// Check if an external error is stored
ELSIF FunctionData.ErrorData.ExternalError.ErrorType > E_ErrorType.NO_ERROR_PENDING THEN
	// If error type has changed - its gone or type has changed
	IF FunctionData.ErrorData.ExternalError.ErrorType <> 
	   FunctionData.ErrorData.Error.ErrorType THEN
	   
		// If the stored error type was "ERROR"
		IF FunctionData.ErrorData.Error.ErrorType = E_ErrorType.ERROR
			OR FunctionData.ErrorData.Error.ErrorType = E_ErrorType.WARNING THEN
			// Send error is gone
			ITC.FunctionITC.Commands.NoErrorReport := TRUE;
		END_IF
		
		// Reset Message
		FunctionData.ErrorData.Error.ResetError 	:= FALSE;
		FunctionData.ErrorData.Error.ErrorType 	:= NO_ERROR_PENDING;
		FunctionData.ErrorData.Error.ErrorCode.Conv:= E_ErrorConv.NO_ERROR_CODE;
		FunctionData.ErrorData.Error.ErrorParam 	:= '';
	END_IF
END_IF

(**************************************************************************************************************
   Check for new or higher prioritized message
***************************************************************************************************************)
// Loop trough all error sets errors 
FOR mIdx := 1 TO NUMBER_OF_ERROR_SETS DO
	// Detect new or higher prioritized error message
	IF FunctionData.ErrorData.ErrorDataSet[mIdx].ErrorType > 
       FunctionData.ErrorData.Error.ErrorType THEN
		// Store index of current data set
		FunctionData.ErrorData.DataSetIdx := mIdx;
		
		// Update error
		FunctionData.ErrorData.Error.ErrorCode.Conv := FunctionData.ErrorData.ErrorDataSet[mIdx].ErrorCode.Conv;
		FunctionData.ErrorData.Error.ErrorParam := FunctionData.ErrorData.ErrorDataSet[mIdx].ErrorParam;
		FunctionData.ErrorData.Error.ErrorType := FunctionData.ErrorData.ErrorDataSet[mIdx].ErrorType;
		
		// Send Report
		ITC.FunctionITC.Commands.StatusReport := TRUE;
	END_IF
	
	// Check is an error is ongoing and a reset command is set
	IF FunctionData.ErrorData.Error.ResetError AND 
       FunctionData.ErrorData.ErrorDataSet[mIdx].ErrorType <> NO_ERROR_PENDING THEN
	   
		// Reset current error data set
		FunctionData.ErrorData.ErrorDataSet[mIdx].ResetError := TRUE;
	END_IF
END_FOR


// Check external error slot
IF FunctionData.ErrorData.ExternalError.ErrorType > FunctionData.ErrorData.Error.ErrorType THEN

	// Reset lower prioritized previous errors
	mDataSetIdx := 0;
	
	// Update error
	FunctionData.ErrorData.Error.ErrorCode.Conv := FunctionData.ErrorData.ExternalError.ErrorCode.Conv;
	FunctionData.ErrorData.Error.ErrorParam := FunctionData.ErrorData.ExternalError.ErrorParam;
	FunctionData.ErrorData.Error.ErrorType := FunctionData.ErrorData.ExternalError.ErrorType;

	// Send Report
	ITC.FunctionITC.Commands.StatusReport := TRUE;
END_IF

// Check is an external error is ongoing and a reset command is set
IF FunctionData.ErrorData.Error.ResetError AND 
   FunctionData.ErrorData.ExternalError.ErrorType <> NO_ERROR_PENDING THEN
   
	// Reset current error data set
	FunctionData.ErrorData.ExternalError.ResetError := TRUE;
END_IF


// If reset command is set
IF FunctionData.ErrorData.Error.ResetError THEN
	// If the stored error type was "ERROR"
	IF FunctionData.ErrorData.Error.ErrorType = E_ErrorType.ERROR THEN
		// Send error is gone
		ITC.FunctionITC.Commands.NoErrorReport := TRUE;
	END_IF
	
	// Reset stored data index
	FunctionData.ErrorData.DataSetIdx := 0;	

	// Reset Message
	FunctionData.ErrorData.Error.ResetError 	:= FALSE;
	FunctionData.ErrorData.Error.ErrorType 	:= NO_ERROR_PENDING;
	FunctionData.ErrorData.Error.ErrorCode.Conv:= E_ErrorConv.NO_ERROR_CODE;
	FunctionData.ErrorData.Error.ErrorParam 	:= '';
END_IF


(**************************************************************************************************************
   Function error state
***************************************************************************************************************)
// If function is in error state
IF FunctionData.ErrorData.Error.ErrorType = E_ErrorType.ERROR THEN
	// Set error state - ERROR
	FunctionData.ErrorData.ErrorState := E_ErrorState.ERROR;
	
// If function is in warning state
ELSIF FunctionData.ErrorData.Error.ErrorType = E_ErrorType.WARNING THEN
	// Set error state - WARNING
	FunctionData.ErrorData.ErrorState := E_ErrorState.WARNING;

// If function has no error or an info is pending
ELSIF FunctionData.ErrorData.Error.ErrorType = E_ErrorType.NO_ERROR_PENDING OR 
	  FunctionData.ErrorData.Error.ErrorType = E_ErrorType.INFO  THEN
	// Set error state - Operational
	FunctionData.ErrorData.ErrorState := E_ErrorState.OPERATIONAL;

ELSE
	// Otherwise -> Unknown
	FunctionData.ErrorData.ErrorState := E_ErrorState.UNKNOWN;
END_IF
END_METHOD

///Monitor zone errors - Verify error handling and report new errors.
METHOD PROTECTED M_MonitorZoneErrors : BOOL
(**************************************************************************************
 * Application   : BoxControl Framework
 * Revision date : $Date: 2021-04-09 16:13:33 +0200 (fre, 09 apr 2021) $
 * Author        : CDC
 * ------------------------------------------------------------------------------------
 * © Swisslog AG * Swisslog is not liable for any usage of this source code that is not agreed
 * on between Swisslog and the other party. The mandatory legal liability remains * unaffected.
 * ------------------------------------------------------------------------------------
 * Project revision history:
 *
 * VERSION DATE         INITIALS     DESCRIPTION
 * 0.0     DD.MM.YYYY   name       	 explain customized modifications
 *
 **************************************************************************************)
VAR
	mDataSetIdx				: INT; // Temporary data set index
	mIdx					: INT; // Iterator
	mZoneIdx				: INT; // Iterator through all zones
END_VAR
// Initialize
FunctionData.ErrorData.ZoneErrorPending := FALSE;

(**************************************************************************************************************
   Zone error handling
***************************************************************************************************************)
// Go through all zones
FOR mZoneIdx := 1 TO SettingsFunction.NumberOfZones DO
	
	// Store current zone data set index
	mDataSetIdx := ZoneData[mZoneIdx].ErrorData.DataSetIdx;
	
	// Check if an error is stored
	IF mDataSetIdx > 0 THEN
		
		// If error type has changed - its gone or type has changed
		IF ZoneData[mZoneIdx].ErrorData.ErrorDataSet[mDataSetIdx].ErrorType <> 
           ZoneData[mZoneIdx].ErrorData.Error.ErrorType THEN
			
			// If the stored error type was "ERROR"
			IF ZoneData[mZoneIdx].ErrorData.Error.ErrorType = E_ErrorType.ERROR
			   OR ZoneData[mZoneIdx].ErrorData.Error.ErrorType = E_ErrorType.WARNING  THEN
				// Send error is gone
				ITC.ZoneITC[mZoneIdx].Commands.NoErrorReport := TRUE;
			END_IF
			
			// Reset stored data index
			ZoneData[mZoneIdx].ErrorData.DataSetIdx := 0;		
					
			// Reset Message
			ZoneData[mZoneIdx].ErrorData.Error.ResetError := FALSE;
			ZoneData[mZoneIdx].ErrorData.Error.ErrorType := NO_ERROR_PENDING;
			ZoneData[mZoneIdx].ErrorData.Error.ErrorCode.Conv := E_ErrorConv.NO_ERROR_CODE;
			ZoneData[mZoneIdx].ErrorData.Error.ErrorParam := '';
		END_IF
		// Check if an external error is stored
	ELSIF ZoneData[mZoneIdx].ErrorData.ExternalError.ErrorType > E_ErrorType.NO_ERROR_PENDING THEN
		// If error type has changed - its gone or type has changed
		IF ZoneData[mZoneIdx].ErrorData.ExternalError.ErrorType <> 
		   ZoneData[mZoneIdx].ErrorData.Error.ErrorType THEN
		   
			// If the stored error type was "ERROR"
			IF ZoneData[mZoneIdx].ErrorData.Error.ErrorType = E_ErrorType.ERROR 
			   OR ZoneData[mZoneIdx].ErrorData.Error.ErrorType = E_ErrorType.WARNING THEN
				// Send error is gone
				ITC.ZoneITC[mZoneIdx].Commands.NoErrorReport := TRUE;
			END_IF
			
			// Reset Message
			ZoneData[mZoneIdx].ErrorData.Error.ResetError 		:= FALSE;
			ZoneData[mZoneIdx].ErrorData.Error.ErrorType 		:= NO_ERROR_PENDING;
			ZoneData[mZoneIdx].ErrorData.Error.ErrorCode.Conv	:= E_ErrorConv.NO_ERROR_CODE;
			ZoneData[mZoneIdx].ErrorData.Error.ErrorParam 		:= '';
		END_IF
	END_IF
	
	(**************************************************************************************************************
	   Check for new or higher prioritized message
	***************************************************************************************************************)
	
	// Loop trough all errors 
	FOR mIdx := 1 TO NUMBER_OF_ERROR_SETS DO
		// Detect new or higher prioritized error message
		IF ZoneData[mZoneIdx].ErrorData.ErrorDataSet[mIdx].ErrorType > 
		   ZoneData[mZoneIdx].ErrorData.Error.ErrorType THEN
			
			// Store index of current data set
			ZoneData[mZoneIdx].ErrorData.DataSetIdx := mIdx;
			
			// Update error
			ZoneData[mZoneIdx].ErrorData.Error.ErrorCode.Conv := ZoneData[mZoneIdx].ErrorData.ErrorDataSet[mIdx].ErrorCode.Conv;
			ZoneData[mZoneIdx].ErrorData.Error.ErrorParam := ZoneData[mZoneIdx].ErrorData.ErrorDataSet[mIdx].ErrorParam;
			ZoneData[mZoneIdx].ErrorData.Error.ErrorType := ZoneData[mZoneIdx].ErrorData.ErrorDataSet[mIdx].ErrorType;
			
			// Send Report
			ITC.ZoneITC[mZoneIdx].Commands.StatusReport := TRUE;
		END_IF
		
		// Check is an error is ongoing and a reset command is set
		IF ZoneData[mZoneIdx].ErrorData.Error.ResetError AND 
		   ZoneData[mZoneIdx].ErrorData.ErrorDataSet[mIdx].ErrorType <> NO_ERROR_PENDING THEN
		   
			// Reset current error data set
			ZoneData[mZoneIdx].ErrorData.ErrorDataSet[mIdx].ResetError := TRUE;
		END_IF
	END_FOR
	
	// Check external error slot
	IF ZoneData[mZoneIdx].ErrorData.ExternalError.ErrorType > ZoneData[mZoneIdx].ErrorData.Error.ErrorType THEN
		// Reset lower prioritized previous errors
		mDataSetIdx := 0;
		
		// Update error
		ZoneData[mZoneIdx].ErrorData.Error.ErrorCode.Conv := ZoneData[mZoneIdx].ErrorData.ExternalError.ErrorCode.Conv;
		ZoneData[mZoneIdx].ErrorData.Error.ErrorParam := ZoneData[mZoneIdx].ErrorData.ExternalError.ErrorParam;
		ZoneData[mZoneIdx].ErrorData.Error.ErrorType := ZoneData[mZoneIdx].ErrorData.ExternalError.ErrorType;
	
		// Send Report
		ITC.ZoneITC[mZoneIdx].Commands.StatusReport := TRUE;
	END_IF
	
	// Check is an external error is ongoing and a reset command is set
	IF ZoneData[mZoneIdx].ErrorData.Error.ResetError AND 
	   ZoneData[mZoneIdx].ErrorData.ExternalError.ErrorType <> NO_ERROR_PENDING THEN
	   
		// Reset current error data set
		ZoneData[mZoneIdx].ErrorData.ExternalError.ResetError := TRUE;
	END_IF
	
	// If reset command is set
	IF ZoneData[mZoneIdx].ErrorData.Error.ResetError THEN

		// If the stored error type was "ERROR"
		IF ZoneData[mZoneIdx].ErrorData.Error.ErrorType = E_ErrorType.ERROR THEN
			// Send error is gone
			ITC.ZoneITC[mZoneIdx].Commands.NoErrorReport := TRUE;
		END_IF
		
		// Reset stored data index
		ZoneData[mZoneIdx].ErrorData.DataSetIdx := 0;	
	
		// Reset Message
		ZoneData[mZoneIdx].ErrorData.Error.ResetError 	:= FALSE;
		ZoneData[mZoneIdx].ErrorData.Error.ErrorType := NO_ERROR_PENDING;
		ZoneData[mZoneIdx].ErrorData.Error.ErrorCode.Conv := E_ErrorConv.NO_ERROR_CODE;
		ZoneData[mZoneIdx].ErrorData.Error.ErrorParam 	:= '';
	END_IF
	
	
	(**************************************************************************************************************
	   zone error state
	***************************************************************************************************************)
	
	// If function is in error state
	IF ZoneData[mZoneIdx].ErrorData.Error.ErrorType = E_ErrorType.ERROR THEN
		// Set error state - ERROR
		ZoneData[mZoneIdx].ErrorData.ErrorState := E_ErrorState.ERROR;
		
	// If function is in warning state
	ELSIF ZoneData[mZoneIdx].ErrorData.Error.ErrorType = E_ErrorType.WARNING THEN
		// Set error state - WARNING
		ZoneData[mZoneIdx].ErrorData.ErrorState := E_ErrorState.WARNING;
	
	// If function has no error or an info is pending
	ELSIF ZoneData[mZoneIdx].ErrorData.Error.ErrorType = E_ErrorType.NO_ERROR_PENDING OR 
		  ZoneData[mZoneIdx].ErrorData.Error.ErrorType = E_ErrorType.INFO  THEN
		// Set error state - Operational
		ZoneData[mZoneIdx].ErrorData.ErrorState := E_ErrorState.OPERATIONAL;
	
	ELSE
		// Otherwise -> Unknown
		ZoneData[mZoneIdx].ErrorData.ErrorState := E_ErrorState.UNKNOWN;
	END_IF
	
	(**************************************************************************************************************
	   Inform function about zone error state
	***************************************************************************************************************)
	FunctionData.ErrorData.ZoneErrorPending := FunctionData.ErrorData.ZoneErrorPending OR
															ZoneData[mZoneIdx].ErrorData.Error.ErrorType = E_ErrorType.ERROR;
END_FOR
END_METHOD

METHOD M_MoveTU_DataIndex : DINT;
(**************************************************************************************
 * 	Application		:	BoxControl Framework
 *	Revision		:	$Revision: 475069 $
 *	Revision date	:	$Date: 2021-04-09 16:13:33 +0200 (fre, 09 apr 2021) $
 *	Last changed by	:	$Author: d7mangc $
 *	URL				:	$URL: http://almscdc.swisslog.com/repo/SWPD/Development/BoxControlFramework/20_Release/tags/R1.12.0/01_Software/BCF/BCF/JumpStart/20_Product/10_BCF/11_Conv/12_E_Functions/FB_FunctionConv.TcPOU $
 *
 *	Purpose			:	Moves the TU-data index from zone to zone and updates the states.
 *
 * ------------------------------------------------------------------------------------
 *	Copyright Swisslog [IP AG], Switzerland. All rights reserved.
 * 
 * ------------------------------------------------------------------------------------
 *	
 * 	Revision History: 
 *
 * 	VERSION			DATE			INITIALS			DESCRIPTION
 *	0.1				01.01.2001		swl					Example
 *
 **************************************************************************************)
VAR_INPUT
	mZoneNumber : INT;
END_VAR
// Return current TU data index
M_MoveTU_dataIndex := ZoneData[mZoneNumber].TransportControlData.TU_DataIndex;
// Update last TU data index
ZoneData[mZoneNumber].TransportControlData.LastTU_DataIndex := M_MoveTU_dataIndex;
// Delete current TU data index
ZoneData[mZoneNumber].TransportControlData.TU_DataIndex := 0;
// Reset data present flag
ZoneData[mZoneNumber].TransportControlData.DataPresent := FALSE;
// Update number of present TUs 
IF ZoneData[mZoneNumber].TransportControlData.NumberOfPresentTUs > 0 THEN
	ZoneData[mZoneNumber].TransportControlData.NumberOfPresentTUs := ZoneData[mZoneNumber].TransportControlData.NumberOfPresentTUs -1;
END_IF


// BCFD-11639 - POR0 - Position Cleared Report sent without TU-ID	
// included in BCF 1.16
// Save data from the last TU for the position clear report
M_SaveDataTU_ZoneLeft (mZoneNumber, M_MoveTU_dataIndex);
END_METHOD

METHOD PROTECTED M_MsgHandlerZone : BOOL
(**************************************************************************************
 * 	Application		:	BoxControl Framework
 *	Revision		:	$Revision: 475069 $
 *	Revision date	:	$Date: 2021-04-09 16:13:33 +0200 (fre, 09 apr 2021) $
 *	Last changed by	:	$Author: d7mangc $
 *	URL				:	$URL: http://almscdc.swisslog.com/repo/SWPD/Development/BoxControlFramework/20_Release/tags/R1.12.0/01_Software/BCF/BCF/JumpStart/20_Product/10_BCF/11_Conv/12_E_Functions/FB_FunctionConv.TcPOU $
 *
 *	Purpose			:	Function zone ITC out interface
 *						Handles internally set ITC commands.
 *
 * ------------------------------------------------------------------------------------
 *	Copyright Swisslog [IP AG], Switzerland. All rights reserved.
 * 
 * ------------------------------------------------------------------------------------
 *	
 * 	Revision History: 
 *
 * 	VERSION			DATE			INITIALS			DESCRIPTION
 *	0.1				01.01.2001		swl					Example
 *
 **************************************************************************************)
VAR_INPUT
	mZoneNumber			: INT; // Zone number	
END_VAR

VAR
	mTU_DataIndex		: DINT;
	mIdx				: INT; // Iterator
END_VAR

// If a valid zone is configured
IF mZoneNumber > 0 AND mZoneNumber <= SettingsFunction.NumberOfZones THEN
	
	// TU data index
	mTU_DataIndex := ZoneData[mZoneNumber].TransportControlData.TU_DataIndex;

	(*******************************************************************************
		Transport Task Complete - TTC
	********************************************************************************)
	// If data are present on zone
	IF ZoneData[mZoneNumber].TransportControlData.DataPresent THEN
		
		// Go through all destination of the TU
		FOR mIdx := 1 TO TU_DataTable[mTU_DataIndex].DataSet.NumberOfDest DO
			// Check destination
			IF TU_DataTable[mTU_DataIndex].Destination[mIdx].eFunctionNumber = SettingsFunction.eFunctionNumber AND
			   TU_DataTable[mTU_DataIndex].Destination[mIdx].ZoneNumber =	mZoneNumber THEN
			   
			   	// When a TTC is requested when data are present
				IF SettingsFunction.Zone[mZoneNumber].SendTransportTaskCompleted AND 
				   NOT ITC.ZoneITC[mZoneNumber].Flags.TransportTaksCompleteSent THEN
					// Send telegram & flag
					ITC.ZoneITC[mZoneNumber].Commands.TransportTaskCompleted := TRUE;
					ITC.ZoneITC[mZoneNumber].Flags.TransportTaksCompleteSent := TRUE;
				END_IF
				
				// When a TTC is requested when data are present and location occupied
				IF SettingsFunction.Zone[mZoneNumber].SendTransportTaskCompletedOcc AND 
				   ZoneData[mZoneNumber].TransportControlData.Occupied AND
				   NOT ITC.ZoneITC[mZoneNumber].Flags.TransportTaksCompleteOccSent THEN
					// Send telegram & flag
					ITC.ZoneITC[mZoneNumber].Commands.TransportTaskCompleted := TRUE;
					ITC.ZoneITC[mZoneNumber].Flags.TransportTaksCompleteOccSent := TRUE;
				END_IF
				
				// When no TTC is configured or already sent - Reset destination
				IF (NOT SettingsFunction.Zone[mZoneNumber].SendTransportTaskCompleted OR ITC.ZoneITC[mZoneNumber].Flags.TransportTaksCompleteSent) AND
				   (NOT SettingsFunction.Zone[mZoneNumber].SendTransportTaskCompletedOcc OR ITC.ZoneITC[mZoneNumber].Flags.TransportTaksCompleteOccSent) THEN
					// Delete destination
					F_DeleteDestination(eFunctionNumber := SettingsFunction.eFunctionNumber, ZoneNumber := mZoneNumber);
				   EXIT;
				END_IF
			END_IF
		END_FOR
	ELSE
		// Reset flags
		ITC.ZoneITC[mZoneNumber].Flags.TransportTaksCompleteSent := FALSE;
		ITC.ZoneITC[mZoneNumber].Flags.TransportTaksCompleteOccSent := FALSE;
	END_IF
	
	(*******************************************************************************
		Position Clear Report 
	********************************************************************************)
	// When a position clear report is requested 
	IF SettingsFunction.Zone[mZoneNumber].SendPositionClear THEN 
		// Is corresponding function started
	   	IF FunctionData.OperationState.eState = E_PositionState.STARTED THEN
			// Is zone free
			IF NOT ZoneData[mZoneNumber].TransportControlData.Occupied THEN
				// And not sent so far
				IF NOT ITC.ZoneITC[mZoneNumber].Flags.PositionClearSent THEN
					// Send telegram & flag
					ITC.ZoneITC[mZoneNumber].Commands.PositionCleared := TRUE;
					ITC.ZoneITC[mZoneNumber].Flags.PositionClearSent := TRUE;
				END_IF
			ELSE
				// Reset flag
				ITC.ZoneITC[mZoneNumber].Flags.PositionClearSent := FALSE;
			END_IF
		END_IF
	ELSE
		// Reset flag
		ITC.ZoneITC[mZoneNumber].Flags.PositionClearSent := FALSE;
	END_IF
	
	(*******************************************************************************
		Position Occupied Report 
	********************************************************************************)
	// When a position occupied report is requested 
	IF SettingsFunction.Zone[mZoneNumber].SendPositionOccupied THEN 
		// Is corresponding function started
	   	IF FunctionData.OperationState.eState = E_PositionState.STARTED THEN
			// Is zone occupied
			IF ZoneData[mZoneNumber].TransportControlData.Occupied THEN
				// And not sent so far
				IF NOT ITC.ZoneITC[mZoneNumber].Flags.PositionOccupiedSent THEN
					// Send telegram & flag
					ITC.ZoneITC[mZoneNumber].Commands.PositionOccupied := TRUE;
					ITC.ZoneITC[mZoneNumber].Flags.PositionOccupiedSent := TRUE;
				END_IF
			ELSE
				// Reset flag
				ITC.ZoneITC[mZoneNumber].Flags.PositionOccupiedSent := FALSE;
			END_IF
		END_IF
	ELSE
		// Reset flag
		ITC.ZoneITC[mZoneNumber].Flags.PositionOccupiedSent := FALSE;
	END_IF
	
	(*******************************************************************************
		Identification Point Report 
	********************************************************************************)
	// When a identification report is requested 
	IF SettingsFunction.Zone[mZoneNumber].SendIdentificationReport THEN 
		// When data are present
		IF ZoneData[mZoneNumber].TransportControlData.DataPresent THEN
			// If the zone is occupied and no add-on is assigned or data ready from all addons is set
			// the telegramm can be triggered.
			IF ZoneData[mZoneNumber].TransportControlData.Occupied THEN 
				IF ZoneData[mZoneNumber].AddOn.NoAddons OR ZoneData[mZoneNumber].AddOn.Orders.DataReady THEN
					// And not sent so far
					IF NOT ITC.ZoneITC[mZoneNumber].Flags.IdentificationReportSent THEN
						// Send telegram & flag
						ITC.ZoneITC[mZoneNumber].Commands.IdentificationReport := TRUE;
						ITC.ZoneITC[mZoneNumber].Flags.IdentificationReportSent := TRUE;
					END_IF
				END_IF
			ELSE
				// Reset flag
				ITC.ZoneITC[mZoneNumber].Flags.IdentificationReportSent := FALSE;
			END_IF
		ELSE
			// Reset flag
			ITC.ZoneITC[mZoneNumber].Flags.IdentificationReportSent := FALSE;
		END_IF
	ELSE
		// Reset flag
		ITC.ZoneITC[mZoneNumber].Flags.IdentificationReportSent := FALSE;
	END_IF
END_IF
END_METHOD

METHOD M_PreInit : BOOL
(**************************************************************************************
 * 	Application		:	BoxControl Framework
 *	Revision		:	$Revision: 475069 $
 *	Revision date	:	$Date: 2021-04-09 16:13:33 +0200 (fre, 09 apr 2021) $
 *	Last changed by	:	$Author: d7mangc $
 *	URL				:	$URL: http://almscdc.swisslog.com/repo/SWPD/Development/BoxControlFramework/20_Release/tags/R1.12.0/01_Software/BCF/BCF/JumpStart/20_Product/10_BCF/11_Conv/12_E_Functions/FB_FunctionConv.TcPOU $
 *
 *	Purpose			:	Preinitialize 
 *						Clears values and load settings
 *
 * ------------------------------------------------------------------------------------
 *	Copyright Swisslog [IP AG], Switzerland. All rights reserved.
 * 
 * ------------------------------------------------------------------------------------
 *	
 * 	Revision History: 
 *
 * 	VERSION			DATE			INITIALS			DESCRIPTION
 *	0.1				01.01.2001		swl					Example
 *
 **************************************************************************************)
VAR
	eFunctionNumber	: E_FunctionNumber; 
	eElementNumber	: E_ElementNumber;
END_VAR
(**************************************************************************************
   		Unregister
***************************************************************************************)	
// If Addon function link has changed
IF SettingsFunction.FunctionLink.eFunctionNumber <> ConfigFunction.FunctionLink.eFunctionNumber AND
   SettingsFunction.FunctionLink.eFunctionNumber > E_FunctionNumber.F_BEGIN_FUNCTION THEN
   
	// Close old addon link
	eFunctionNumber := SettingsFunction.FunctionLink.eFunctionNumber;
	
	// Is this reference valid
	IF __ISVALIDREF(FunctionRegistry[eFunctionNumber].rFunction) THEN
		// Close AddOn link
		FunctionRegistry[eFunctionNumber].rFunction.M_CloseAddOnLink(eAddOnNumber := SettingsFunction.eFunctionNumber);
	END_IF
END_IF

// If element link has changed
IF SettingsFunction.eElementLink <> ConfigFunction.eElementLink AND 
   SettingsFunction.eElementLink > E_ElementNumber.E_BEGIN_ELEMENT THEN
	// Close old element link
	eElementNumber := SettingsFunction.eElementLink;
	
	// Is reference valid
	IF __ISVALIDREF(ElementRegistry[eElementNumber].rElement) THEN
		// Unregister function in element
		ElementRegistry[eElementNumber].rElement.M_CloseElementLink(SettingsFunction.eFunctionNumber);
	END_IF
END_IF


// Clear previous and next function
FunctionInterface.In.ePrevFunctionNumber := E_FunctionNumber.F_BEGIN_FUNCTION;
FunctionInterface.In.eNextFunctionNumber := E_FunctionNumber.F_BEGIN_FUNCTION;


(**************************************************************************************
	Load 
***************************************************************************************)
SettingsFunction := ConfigFunction;
END_METHOD

METHOD PROTECTED M_ProcessAddOns
(**************************************************************************************
 * 	Application		:	BoxControl Framework
 *	Revision		:	$Revision: 475069 $
 *	Revision date	:	$Date: 2021-04-09 16:13:33 +0200 (fre, 09 apr 2021) $
 *	Last changed by	:	$Author: d7mangc $
 *	URL				:	$URL: http://almscdc.swisslog.com/repo/SWPD/Development/BoxControlFramework/20_Release/tags/R1.12.0/01_Software/BCF/BCF/JumpStart/20_Product/10_BCF/11_Conv/12_E_Functions/FB_FunctionConv.TcPOU $
 *
 *	Purpose			:	Process AddOns
 *
 * ------------------------------------------------------------------------------------
 *	Copyright Swisslog [IP AG], Switzerland. All rights reserved.
 * 
 * ------------------------------------------------------------------------------------
 *	
 * 	Revision History: 
 *
 * 	VERSION			DATE			INITIALS			DESCRIPTION
 *	0.1				01.01.2001		swl					Example
 *
 **************************************************************************************)
VAR
  mIdx             : INT; // Iterator
  mZoneNumber      : INT; // Zone number
  mTU_DataIndexNew : DINT; // TU data index new
  mTU_DataIndexOld : DINT; // TU data index old
  mSummary         : ST_AddOnOrders;
END_VAR
// Initialize var
mSummary.Enable         	:= TRUE;
mSummary.EnableHandover 	:= TRUE;
mSummary.EnableTakeover 	:= TRUE;
mSummary.DataReady      	:= TRUE;
mSummary.TU_DataIndex   	:= 0;
mSummary.EnableSimultaneousTransport := FALSE;
mSummary.UseOwnSensor 		:= FALSE;
mSummary.AddOnSensor 		:= FALSE;
mSummary.AllowDriveTakeover := FALSE;
mSummary.AllowDriveHandover := FALSE;

// Initialize all zones
FOR mIdx := 1 TO SettingsFunction.NumberOfZones DO
	ZoneData[mIdx].AddOn.NoAddons := TRUE;
	ZoneData[mIdx].AddOn.Orders := mSummary;
END_FOR

// Initialize function
FunctionData.AddOn.NoAddons := TRUE;
FunctionData.AddOn.Orders := mSummary;

// Build summary of all addon functions
FOR mIdx := 1 TO NUMBER_OF_ADDON_FUNCTIONS DO
	// If no addon is configured
	IF FunctionInterface.In.AddOnOrder[mIdx].eFunctionNumber = E_FunctionNumber.F_BEGIN_FUNCTION THEN
		// Exit loop
		EXIT;
	END_IF

	// Update summary from addon interface		   
	IF NOT FunctionInterface.In.AddOnOrder[mIdx].Orders.Enable THEN
		mSummary.Enable := FALSE;
	END_IF
	
	IF NOT FunctionInterface.In.AddOnOrder[mIdx].Orders.EnableHandover THEN
		mSummary.EnableHandover := FALSE;
	END_IF

	IF NOT FunctionInterface.In.AddOnOrder[mIdx].Orders.EnableTakeover  THEN
		mSummary.EnableTakeover := FALSE;
	END_IF

	IF NOT FunctionInterface.In.AddOnOrder[mIdx].Orders.DataReady THEN
		mSummary.DataReady := FALSE;
	END_IF
	
	IF NOT FunctionInterface.In.AddOnOrder[mIdx].Orders.DataValid THEN
		mSummary.DataValid := FALSE;
	END_IF
			
    IF FunctionInterface.In.AddOnOrder[mIdx].Orders.EnableSimultaneousTransport THEN
        mSummary.EnableSimultaneousTransport := TRUE;
	END_IF
    
    IF FunctionInterface.In.AddOnOrder[mIdx].Orders.AddOnSensor THEN
        mSummary.AddOnSensor := TRUE;
	END_IF
    
    IF FunctionInterface.In.AddOnOrder[mIdx].Orders.UseOwnSensor THEN
        mSummary.UseOwnSensor := TRUE;
	END_IF
    
    IF FunctionInterface.In.AddOnOrder[mIdx].Orders.AllowDriveTakeover THEN
        mSummary.AllowDriveTakeover := TRUE;
	END_IF
    
    IF FunctionInterface.In.AddOnOrder[mIdx].Orders.AllowDriveHandover THEN
        mSummary.AllowDriveHandover := TRUE;
	END_IF
    
	// Update zone or function data
	mZoneNumber := FunctionInterface.In.AddOnOrder[mIdx].ZoneNumber;
	
	IF mZoneNumber <= 0 THEN
		FunctionData.AddOn.NoAddons := FALSE;
		FunctionData.AddOn.Orders := mSummary;
	ELSIF mZoneNumber > SettingsFunction.NumberOfZones  THEN
		FunctionData.AddOn.NoAddons := FALSE;
		FunctionData.AddOn.Orders := mSummary;
	ELSE
		ZoneData[mZoneNumber].AddOn.NoAddons := FALSE;
		ZoneData[mZoneNumber].AddOn.Orders := mSummary;
	END_IF

	// If it is not a function type "Scanner"
	IF FunctionInterface.In.AddOnOrder[mIdx].eFunctionType <> E_FunctionType.Scanner THEN
		// Process next addon function
		CONTINUE;
	END_IF
	
	// Data ready is not set
	IF NOT FunctionInterface.In.AddOnOrder[mIdx].Orders.DataReady THEN
		// Process next addon function
		CONTINUE;
	END_IF
	
	// Data valid is not set
	IF NOT FunctionInterface.In.AddOnOrder[mIdx].Orders.DataValid THEN
		// Process next addon function
		CONTINUE;
	END_IF

	// Take over TU index
	mTU_DataIndexOld := ZoneData[mZoneNumber].TransportControlData.TU_DataIndex;
	mTU_DataIndexNew := FunctionInterface.In.AddOnOrder[mIdx].Orders.TU_DataIndex;
	ZoneData[mZoneNumber].AddOn.Orders.TU_DataIndex := mTU_DataIndexNew;

	// Update index only if takeover is active, feedin or multi TU	
	IF (ZoneData[mZoneNumber].TransportControlData.eTakeOverState = E_TakeOverState.ACTIVE AND
		(ZoneData[mZoneNumber].TransportControlData.eTransportState = E_TransportState.TAKEOVER OR
		 ZoneData[mZoneNumber].TransportControlData.eTransportState = E_TransportState.SIMULTANEOUS)) OR
	   ZoneData[mZoneNumber].TransportControlData.eTransportState = E_TransportState.FEEDIN OR
	   ZoneData[mZoneNumber].TransportControlData.eTransportState = E_TransportState.MULTI_TU THEN

		// When the conveyor do not have an index yet, just apply the scanner index
		IF mTU_DataIndexOld = 0 THEN
			// Create debug message	
			// '11-001-0095-01-1,  TU_DataIndex inserted by scanner,  TU_DataIndex = 5,  TuID = 000012345,  AssignmentID = 999999999 '
			DebugMsg := '';
			DebugMsg := CONCAT(DebugMsg, F_AddDividerToSisString(SettingsFunction.Zone[mZoneNumber].ZoneName));
			DebugMsg := CONCAT(DebugMsg, ',  TU_DataIndex inserted by scanner');
			DebugMsg := CONCAT(DebugMsg, F_CreateTU_DataString(TU_DataIndex:= mTU_DataIndexNew));
			fbDebugMsg.M_SendInfoMsg(DebugMsg);

			// Update TU data index
			ZoneData[mZoneNumber].TransportControlData.LastTU_DataIndex := mTU_DataIndexOld;
			ZoneData[mZoneNumber].TransportControlData.TU_DataIndex := mTU_DataIndexNew;
			ZoneData[mZoneNumber].TransportControlData.DataPresent := mTU_DataIndexNew <> 0;
	
			// Update current TU position
			TU_DataTable[mTU_DataIndexNew].CurrentFunctionNumber := SettingsFunction.eFunctionNumber;
			TU_DataTable[mTU_DataIndexNew].CurrentZoneNumber := mZoneNumber;

		// When a scanner provides an index unequal to the already existing conveyor index, takeover the scanner index.
		ELSIF mTU_DataIndexOld <> mTU_DataIndexNew THEN
			// Create debug message	
			// '11-001-0095-01-1,  TU_DataIndex overwritten by scanner (old/new),  TU_DataIndex = 5,  TuID = 000012345,  AssignmentID = 999999999,  TU_DataIndex = 9,  TuID = 000098765,  AssignmentID = 999999999',  Origin = 11-002-0125-02-2
			DebugMsg := '';
			DebugMsg := CONCAT(DebugMsg, F_AddDividerToSisString(SettingsFunction.Zone[mZoneNumber].ZoneName));
			DebugMsg := CONCAT(DebugMsg, ',  TU_DataIndex overwritten by scanner (old/new)');
			DebugMsg := CONCAT(DebugMsg, F_CreateTU_DataString(TU_DataIndex:= mTU_DataIndexOld));
			DebugMsg := CONCAT(DebugMsg, F_CreateTU_DataString(TU_DataIndex:= mTU_DataIndexNew));
			DebugMsg := CONCAT(DebugMsg, DebugTextBlocks.ORIGIN);
			DebugMsg := CONCAT(DebugMsg, F_GetFunctionName(
												eFunctionNumber := TU_DataTable[mTU_DataIndexNew].CurrentFunctionNumber,
												ZoneNumber := TU_DataTable[mTU_DataIndexNew].CurrentZoneNumber));
			fbDebugMsg.M_SendErrorMsg(DebugMsg);
												
			// If old TU data index is unknown, delete it from the table 
			IF TU_DataTable[mTU_DataIndexOld].TU_ID.ASCII = Conveyor.TU_ID_UNKNOWN THEN
				// debug message: '11-001-0095-01-1,  unknown old TU_DataIndex deleted,  TU_DataIndex = 5,  TuID = 000012345,  AssignmentID = 999999999'
				DebugMsg := '';
				DebugMsg := CONCAT(DebugMsg, F_AddDividerToSisString(SettingsFunction.Zone[mZoneNumber].ZoneName));
				DebugMsg := CONCAT(DebugMsg, ',  unknown old TU_DataIndex deleted');
				DebugMsg := CONCAT(DebugMsg, F_CreateTU_DataString(TU_DataIndex:= mTU_DataIndexOld));
				fbDebugMsg.M_SendErrorMsg(DebugMsg);
				// Delete data set
				F_DeleteTU_Data(TU_DataIndex := mTU_DataIndexOld,
                       			NoTTC := FALSE);
			END_IF

			// Update TU data index
			ZoneData[mZoneNumber].TransportControlData.LastTU_DataIndex := mTU_DataIndexOld;
			ZoneData[mZoneNumber].TransportControlData.TU_DataIndex := mTU_DataIndexNew;
			ZoneData[mZoneNumber].TransportControlData.DataPresent := mTU_DataIndexNew <> 0;
	
			// Update current TU position
			TU_DataTable[mTU_DataIndexNew].CurrentFunctionNumber := SettingsFunction.eFunctionNumber;
			TU_DataTable[mTU_DataIndexNew].CurrentZoneNumber := mZoneNumber;
		END_IF
					   
    	// Send ACK
		F_AckAddon(eFunctionNumber := FunctionInterface.In.AddOnOrder[mIdx].eFunctionNumber);
						
	ELSIF ZoneData[mZoneNumber].TransportControlData.eTransportState = E_TransportState.HANDOVER OR
		  ZoneData[mZoneNumber].TransportControlData.eTransportState = E_TransportState.OCCUPIED THEN
		 // Send ACK
		F_AckAddon(eFunctionNumber := FunctionInterface.In.AddOnOrder[mIdx].eFunctionNumber);
	END_IF
END_FOR
END_METHOD

METHOD M_ResetError : BOOL
(**************************************************************************************
 * 	Application		:	BoxControl Framework
 *	Revision		:	$Revision: 475069 $
 *	Revision date	:	$Date: 2021-04-09 16:13:33 +0200 (fre, 09 apr 2021) $
 *	Last changed by	:	$Author: d7mangc $
 *	URL				:	$URL: http://almscdc.swisslog.com/repo/SWPD/Development/BoxControlFramework/20_Release/tags/R1.12.0/01_Software/BCF/BCF/JumpStart/20_Product/10_BCF/11_Conv/12_E_Functions/FB_FunctionConv.TcPOU $
 *
 *	Purpose			:	Reset function or zone errors.
 *
 * ------------------------------------------------------------------------------------
 *	Copyright Swisslog [IP AG], Switzerland. All rights reserved.
 * 
 * ------------------------------------------------------------------------------------
 *	
 * 	Revision History: 
 *
 * 	VERSION			DATE			INITIALS			DESCRIPTION
 *	0.1				01.01.2001		swl					Example
 *
 **************************************************************************************)
VAR_INPUT
	mZoneNumber		: INT; // Zone number
	mResetAll		: BOOL; // Reset all
END_VAR

VAR
	mIdx			: INT; // Iterator
END_VAR
// Command is to reset all
IF mResetAll THEN
	// Go through all zones
	FOR mIdx := 1 TO NUMBER_OF_ZONES_PER_FUNCTION DO
		// If the zone is in error
		IF ZoneData[mIdx].ErrorData.Error.ErrorType  <> E_ErrorType.NO_ERROR_PENDING  THEN
			// Send reset
			ZoneData[mIdx].ErrorData.Error.ResetError := TRUE;
		END_IF
	END_FOR

	// If the function is in error
	IF FunctionData.ErrorData.Error.ErrorType  <> E_ErrorType.NO_ERROR_PENDING  THEN
		// Send reset
		FunctionData.ErrorData.Error.ResetError := TRUE;
	END_IF
	
// Command to reset a zone
ELSIF mZoneNumber > 0 AND mZoneNumber <= NUMBER_OF_ZONES_PER_FUNCTION THEN
	// If the zone is in error
	IF ZoneData[mZoneNumber].ErrorData.Error.ErrorType  <> E_ErrorType.NO_ERROR_PENDING  THEN
		// Send reset
		ZoneData[mZoneNumber].ErrorData.Error.ResetError := TRUE;
	END_IF
ELSE
	// If the function is in error
	IF FunctionData.ErrorData.Error.ErrorType  <> E_ErrorType.NO_ERROR_PENDING  THEN
		// Send reset
		FunctionData.ErrorData.Error.ResetError := TRUE;
	END_IF
END_IF

M_ResetError := TRUE;
END_METHOD

METHOD M_ResetExternalError : BOOL
(**************************************************************************************
 * 	Application		:	BoxControl Framework
 *	Revision		:	$Revision: 475069 $
 *	Revision date	:	$Date: 2021-04-09 16:13:33 +0200 (fre, 09 apr 2021) $
 *	Last changed by	:	$Author: d7mangc $
 *	URL				:	$URL: http://almscdc.swisslog.com/repo/SWPD/Development/BoxControlFramework/20_Release/tags/R1.12.0/01_Software/BCF/BCF/JumpStart/20_Product/10_BCF/11_Conv/12_E_Functions/FB_FunctionConv.TcPOU $
 *
 *	Purpose			:	Reset external error
 *						
 *
 * ------------------------------------------------------------------------------------
 *	Copyright Swisslog [IP AG], Switzerland. All rights reserved.
 * 
 * ------------------------------------------------------------------------------------
 *	
 * 	Revision History: 
 *
 * 	VERSION			DATE			INITIALS			DESCRIPTION
 *	0.1				01.01.2001		swl					Example
 *
 **************************************************************************************)
 VAR_INPUT
	mZoneNumber	: INT; // Related zone, 0 = Function itself
	mReset		: BOOL; // Force reset
END_VAR
// Initialize
M_ResetExternalError := FALSE;

IF mZoneNumber > 0 THEN
	// Reset error if ResetError command or reset command is set 
	IF ZoneData[mZoneNumber].ErrorData.ExternalError.ResetError OR mReset THEN
		// Clear error
		ZoneData[mZoneNumber].ErrorData.ExternalError.ResetError 		:= FALSE; 
		ZoneData[mZoneNumber].ErrorData.ExternalError.ErrorType 		:= NO_ERROR_PENDING;
		ZoneData[mZoneNumber].ErrorData.ExternalError.ErrorCode.Conv	:= E_ErrorConv.NO_ERROR_CODE;
		ZoneData[mZoneNumber].ErrorData.ExternalError.ErrorParam 		:= '';
		M_ResetExternalError 								:= TRUE;
	END_IF
ELSE
	// Reset error if ResetError command or reset command is set 
	IF FunctionData.ErrorData.ExternalError.ResetError OR mReset THEN
		// Clear error
		FunctionData.ErrorData.ExternalError.ResetError 	:= FALSE; 
		FunctionData.ErrorData.ExternalError.ErrorType 		:= NO_ERROR_PENDING;
		FunctionData.ErrorData.ExternalError.ErrorCode.Conv	:= E_ErrorConv.NO_ERROR_CODE;
		FunctionData.ErrorData.ExternalError.ErrorParam 	:= '';
		M_ResetExternalError 								:= TRUE;
	END_IF
END_IF
END_METHOD

METHOD PUBLIC M_SaveDataTU_ZoneLeft : BOOL
VAR_INPUT
	mZoneNumber		: INT;
    mTU_DataIndex	: DINT;
END_VAR

// BCFD-11639 - POR0 - Position Cleared Report sent without TU-ID	
// included in BCF 1.16

// Save data from the last TU for the position clear report
ZoneData[mZoneNumber].LastTUdata.AssignmentID	:= TU_DataTable[mTU_DataIndex].AssignmentID;
ZoneData[mZoneNumber].LastTUdata.TU_ID			:= TU_DataTable[mTU_DataIndex].TU_ID.ASCII;
ZoneData[mZoneNumber].LastTUdata.TU_Type		:= TU_DataTable[mTU_DataIndex].DataSet.TU_Type;
END_METHOD

METHOD M_SetEnableHandOver : BOOL
(**************************************************************************************
 * 	Application		:	BoxControl Framework
 *	Revision		:	$Revision: 475069 $
 *	Revision date	:	$Date: 2021-04-09 16:13:33 +0200 (fre, 09 apr 2021) $
 *	Last changed by	:	$Author: d7mangc $
 *	URL				:	$URL: http://almscdc.swisslog.com/repo/SWPD/Development/BoxControlFramework/20_Release/tags/R1.12.0/01_Software/BCF/BCF/JumpStart/20_Product/10_BCF/11_Conv/12_E_Functions/FB_FunctionConv.TcPOU $
 *
 *	Purpose			:	Initialize base functionality of function.
 *
 * ------------------------------------------------------------------------------------
 *	Copyright Swisslog [IP AG], Switzerland. All rights reserved.
 * 
 * ------------------------------------------------------------------------------------
 *	
 * 	Revision History: 
 *
 * 	VERSION			DATE			INITIALS			DESCRIPTION
 *	0.1				01.01.2001		swl					Example
 *
 **************************************************************************************)
VAR_INPUT
	mZoneNumber 	: INT; // Zone number
	mValue			: BOOL; // Set/reset value
END_VAR
// If zone number is valid
IF mZoneNumber > 0 AND mZoneNumber <= SettingsFunction.NumberOfZones THEN
	// Modify variable
	ZoneInterface[mZoneNumber].In.Enable.HandOver := mValue;
	M_SetEnableHandOver := TRUE;

// Otherwise requested index was not found
ELSE	
	DebugMsg := CONCAT('Requested zone not available: ', INT_TO_STRING(mZoneNumber));
	fbDebugMsg.M_SendErrorMsg(DebugMsg);
END_IF
END_METHOD

METHOD M_SetEnableTakeOver : BOOL
(**************************************************************************************
 * 	Application		:	BoxControl Framework
 *	Revision		:	$Revision: 475069 $
 *	Revision date	:	$Date: 2021-04-09 16:13:33 +0200 (fre, 09 apr 2021) $
 *	Last changed by	:	$Author: d7mangc $
 *	URL				:	$URL: http://almscdc.swisslog.com/repo/SWPD/Development/BoxControlFramework/20_Release/tags/R1.12.0/01_Software/BCF/BCF/JumpStart/20_Product/10_BCF/11_Conv/12_E_Functions/FB_FunctionConv.TcPOU $
 *
 *	Purpose			:	Initialize base functionality of function.
 *
 * ------------------------------------------------------------------------------------
 *	Copyright Swisslog [IP AG], Switzerland. All rights reserved.
 * 
 * ------------------------------------------------------------------------------------
 *	
 * 	Revision History: 
 *
 * 	VERSION			DATE			INITIALS			DESCRIPTION
 *	0.1				01.01.2001		swl					Example
 *
 **************************************************************************************)
VAR_INPUT
	mZoneNumber 	: INT; // Zone number
	mValue			: BOOL; // Set/reset value
END_VAR
// If zone number is valid
IF mZoneNumber > 0 AND mZoneNumber <= SettingsFunction.NumberOfZones THEN
	// Modify variable
	ZoneInterface[mZoneNumber].In.Enable.TakeOver := mValue;
	M_SetEnableTakeOver := TRUE;

// Otherwise requested index was not found
ELSE	
	DebugMsg := CONCAT('Requested zone not available: ', INT_TO_STRING(mZoneNumber));
	fbDebugMsg.M_SendErrorMsg(DebugMsg);
END_IF
END_METHOD

METHOD M_SetEnableTransport : BOOL
(**************************************************************************************
 * 	Application		:	BoxControl Framework
 *	Revision		:	$Revision: 475069 $
 *	Revision date	:	$Date: 2021-04-09 16:13:33 +0200 (fre, 09 apr 2021) $
 *	Last changed by	:	$Author: d7mangc $
 *	URL				:	$URL: http://almscdc.swisslog.com/repo/SWPD/Development/BoxControlFramework/20_Release/tags/R1.12.0/01_Software/BCF/BCF/JumpStart/20_Product/10_BCF/11_Conv/12_E_Functions/FB_FunctionConv.TcPOU $
 *
 *	Purpose			:	Initialize base functionality of function.
 *
 * ------------------------------------------------------------------------------------
 *	Copyright Swisslog [IP AG], Switzerland. All rights reserved.
 * 
 * ------------------------------------------------------------------------------------
 *	
 * 	Revision History: 
 *
 * 	VERSION			DATE			INITIALS			DESCRIPTION
 *	0.1				01.01.2001		swl					Example
 *
 **************************************************************************************)
VAR_INPUT
	mZoneNumber 	: INT; // Zone number
	mValue			: BOOL; // Set/reset value
END_VAR
// If zone number is valid
IF mZoneNumber > 0 AND mZoneNumber <= SettingsFunction.NumberOfZones THEN
	// Modify variable
	ZoneInterface[mZoneNumber].In.Enable.Transport := mValue;
	M_SetEnableTransport := TRUE;

// Otherwise requested index was not found
ELSE	
	DebugMsg := CONCAT('Requested zone not available: ', INT_TO_STRING(mZoneNumber));
	fbDebugMsg.M_SendErrorMsg(DebugMsg);
END_IF
END_METHOD

METHOD M_SetExternalError : BOOL
(**************************************************************************************
 * 	Application		:	BoxControl Framework
 *	Revision		:	$Revision: 475069 $
 *	Revision date	:	$Date: 2021-04-09 16:13:33 +0200 (fre, 09 apr 2021) $
 *	Last changed by	:	$Author: d7mangc $
 *	URL				:	$URL: http://almscdc.swisslog.com/repo/SWPD/Development/BoxControlFramework/20_Release/tags/R1.12.0/01_Software/BCF/BCF/JumpStart/20_Product/10_BCF/11_Conv/12_E_Functions/FB_FunctionConv.TcPOU $
 *
 *	Purpose			:	Set error
 *						Wrapped to a function to improve debugging and readability.
 *						
 *
 * ------------------------------------------------------------------------------------
 *	Copyright Swisslog [IP AG], Switzerland. All rights reserved.
 * 
 * ------------------------------------------------------------------------------------
 *	
 * 	Revision History: 
 *
 * 	VERSION			DATE			INITIALS			DESCRIPTION
 *	0.1				01.01.2001		swl					Example
 *
 **************************************************************************************)
 VAR_INPUT
	mZoneNumber		: INT; // Related zone, 0 = Function itself
	mErrorType		: E_ErrorType; // Error message type
	mErrorParam		: STRING(System.ERROR_PARAM_STRINGLENGTH); // Error parameter
	mErrorCode		: INT; // Error message
END_VAR
// Initialize
M_SetExternalError := FALSE;

// Check that the values are valid
IF mErrorType > E_ErrorType.NO_ERROR_PENDING AND mErrorCode > E_ErrorConv.NO_ERROR_CODE THEN
	IF mZoneNumber > 0 THEN
		ZoneData[mZoneNumber].ErrorData.ExternalError.ErrorCode.Conv := mErrorCode;
		ZoneData[mZoneNumber].ErrorData.ExternalError.ErrorType := mErrorType;
		ZoneData[mZoneNumber].ErrorData.ExternalError.ErrorParam := mErrorParam;
	ELSE
		FunctionData.ErrorData.ExternalError.ErrorCode.Conv := mErrorCode;
		FunctionData.ErrorData.ExternalError.ErrorType := mErrorType;
		FunctionData.ErrorData.ExternalError.ErrorParam := mErrorParam;
	END_IF
	
	M_SetExternalError := TRUE;
END_IF
END_METHOD

METHOD M_UpdateRegistry
(**************************************************************************************
 * 	Application		:	BoxControl Framework
 *	Revision		:	$Revision: 475069 $
 *	Revision date	:	$Date: 2021-04-09 16:13:33 +0200 (fre, 09 apr 2021) $
 *	Last changed by	:	$Author: d7mangc $
 *	URL				:	$URL: http://almscdc.swisslog.com/repo/SWPD/Development/BoxControlFramework/20_Release/tags/R1.12.0/01_Software/BCF/BCF/JumpStart/20_Product/10_BCF/11_Conv/12_E_Functions/FB_FunctionConv.TcPOU $
 *
 *	Purpose			:	Update registry information
 *
 * ------------------------------------------------------------------------------------
 *	Copyright Swisslog [IP AG], Switzerland. All rights reserved.
 * 
 * ------------------------------------------------------------------------------------
 *	
 * 	Revision History: 
 *
 * 	VERSION			DATE			INITIALS			DESCRIPTION
 *	0.1				01.01.2001		swl					Example
 *
 **************************************************************************************)
VAR_INPUT
END_VAR
VAR
	mIdx	: INT;
END_VAR

IF ConfigFunction.eFunctionNumber > E_FunctionNumber.F_BEGIN_FUNCTION THEN

	FunctionRegistry[ConfigFunction.eFunctionNumber].rFunctionData REF= FunctionData;
	FunctionRegistry[ConfigFunction.eFunctionNumber].rFunctionInterface REF= FunctionInterface;
	FunctionRegistry[ConfigFunction.eFunctionNumber].rSettingsFunction REF= SettingsFunction;
	FOR mIdx := 1 TO ConfigFunction.NumberOfZones DO
		FunctionRegistry[ConfigFunction.eFunctionNumber].Zone[mIdx].refZoneData REF= ZoneData[mIdx];
		FunctionRegistry[ConfigFunction.eFunctionNumber].Zone[mIdx].refZoneInterface REF= ZoneInterface[mIdx];
	END_FOR
END_IF
END_METHOD

END_FUNCTION_BLOCK

(* stored: Version 1.1.0.1, ProductVersion 3.1.4024.9
   POU FB_FunctionConv: Id {59c4c264-1ea2-492c-8cba-53173e028310}, SpecialFunc None
   Action A_ErrorHandler: Id {f04b2c14-5d9b-48b2-8c20-a29b993700a3}
   Action A_StateControl: Id {6bf0f59b-d533-4912-8197-1b83e5bbd1f8}
   Method FB_init: Id {93e6baa7-6db1-4292-bf48-7fd5b0e30131}
   Method M_AddOnAck: Id {a8dfbd28-af97-4152-9cbb-19bc5d1b1328}
   Method M_CloseAddOnLink: Id {0cd96de5-3e46-4ec4-9164-d7f42e41b5d9}
   Method M_CreateAddOnLink: Id {52b3cec9-4297-40d7-988a-984ec97ea48d}
   Method M_DeleteTU_DataIndex: Id {8f0cbd51-7359-4826-ba2a-8aec90b7752b}
   Method M_FindTU_DataIndex: Id {bd46c852-9938-4845-9e47-705427d1c5d0}
   Method M_GetAddOnOrder: Id {c2b8a265-7e1e-43ff-9a46-f88bd0c658e5}
   Method M_GetElementStates: Id {d6acfe2a-4cd5-4de2-bbf6-d707853bce1f}
   Method M_GetNextTransportData: Id {5ced4e8b-1275-48c3-a54b-2c99c75bd265}
   Method M_GetOutAddOnOrders: Id {cde65947-0af5-4c31-97f6-4fa11a9073b5}
   Method M_GetPreviousTransportData: Id {586344ff-2bc2-4340-b5ce-7ce98897ed1d}
   Method M_GetTransportControlParam: Id {495d7719-427a-4540-b7d6-d36a41acf0c2}
   Method M_GetTransportData: Id {ad17fd6b-3b62-4afb-a203-7ee2d6bdaca3}
   Method M_InitFunction: Id {3e2d2066-15cd-4fb8-8f14-4baf31a3197a}
   Method M_ITC_AddTU_Data: Id {1cd622f1-30bb-4d21-9d90-c65c9db38cef}
   Method M_ITC_DAQ: Id {a9e43913-fe27-4d33-ba4e-8e2c644ede31}
   Method M_ITC_DataAquisitionZone: Id {7df87bd1-4872-4b78-8353-43b011e81eb8}
   Method M_ITC_FCQ: Id {27776317-a1e1-4d55-88b1-c913d79b8ece}
   Method M_ITC_FSQ: Id {cf04fb33-e1ee-4bda-9d8b-da92b0dff3c1}
   Method M_ITC_GDQ: Id {9a21e5c4-62d7-49f2-8d14-eb246db5e801}
   Method M_ITC_MCQ: Id {ac22eb88-b611-4d1c-963d-f1f60e354500}
   Method M_ITC_ProcessMsg: Id {3446d6e6-ff2b-47b2-9683-db16bac5e938}
   Method M_ITC_ProcessOut: Id {a0f13611-81b8-4609-854b-98ed9fb4410d}
   Method M_ITC_ProcessOutZone: Id {037a2786-fddd-481e-8584-8492e5eaec32}
   Method M_ITC_RAA: Id {b9c4e0e7-a8c7-4992-a22c-2c6713d06f4f}
   Method M_ITC_RDQ: Id {d074124b-d2dd-4238-8911-401815057041}
   Method M_ITC_SIQ: Id {c85d9a78-b4ae-402e-8cd4-a561e9aa74a7}
   Method M_MonitorFunctionErrors: Id {0ec46405-bab9-4f19-9d28-837931958e3a}
   Method M_MonitorZoneErrors: Id {3306cd3a-bf44-4db9-b1e2-edf22bbbc7bc}
   Method M_MoveTU_DataIndex: Id {3bb46781-798e-4364-911b-1fb174d9dc11}
   Method M_MsgHandlerZone: Id {6a3e4055-94c9-4b38-b363-45c8c4cfb575}
   Method M_PreInit: Id {4e42ab4a-6eab-4421-a7e5-5f2fbc031833}
   Method M_ProcessAddOns: Id {38fde08f-241b-4873-9821-2435792365a9}
   Method M_ResetError: Id {bc8d095b-6de7-4a09-bde9-10d11dfa72cd}
   Method M_ResetExternalError: Id {9b9adaa3-012d-4c65-8033-fde76c862120}
   Method M_SaveDataTU_ZoneLeft: Id {1855497e-8420-4ffe-b372-d5b83aff6858}
   Method M_SetEnableHandOver: Id {4cc339a4-c5a2-497e-9e35-a2db1d902116}
   Method M_SetEnableTakeOver: Id {b817cf1d-ed45-4e0f-be7a-08f27bdb1f84}
   Method M_SetEnableTransport: Id {984725c7-90f4-407e-b34e-2d0308138985}
   Method M_SetExternalError: Id {ac71b258-fd95-43a7-bc7b-3b4793cc8a29}
   Method M_UpdateRegistry: Id {cc96d081-f5de-4643-a164-040bd0f9ebe9} *)
